INTERFACE ITF_Control2_HMI_Init EXTENDS ITF_BaseControlElement, ITF_Control2_HMI_Connector

END_INTERFACE

(* stored: Version 1.1.0.1
   Itf ITF_Control2_HMI_Init: Id {b1cbdee3-d421-0d53-3e42-7fdeb8db61fe} *)
